(*
SPDX-FileCopyrightText: © 2026 Oleksandr Tiutyk <trofimich@gmail.com>
SPDX-License-Identifier: MIT
License: https://opensource.org/license/mit
*)

(*!
<summary>Executes TryActivity and recovers via an optional CatchActivity when TryActivity raises an exception.</summary>
<description>
When TryActivity throws a non-terminal exception and CatchActivity is configured, synchronous diagnostics are
passed to CatchActivity.CaptureException before starting CatchActivity. Terminal allocation failures and
exceptions when CatchActivity is 0 (or thrown by CatchActivity itself) propagate to the parent. Resetting
resets both TryActivity and CatchActivity back to PASSIVE_READY and clears CurrentActivity. Catch startup
does not wait for asynchronous cleanup in the failed try branch. The recovery implementation must use
independent resources or explicitly coordinate cleanup completion before reusing a shared resource.
A failed try branch is not automatically reset before catch. After the composite finishes, RequestReset
provides the ordinary path for driving pending cancellation/reset work before a fresh run.
</description>
*)

{attribute 'no_explicit_call' := 'do not call this function block directly'}
{attribute 'enable_dynamic_creation'}
FUNCTION_BLOCK TryCatchActivity EXTENDS ExclusiveCompositeActivity
	IMPLEMENTS ITryCatchActivity, TOF_Core.IConfigurationSerializable
VAR_STAT
	{attribute 'hide'}
	_ClassName : STRING := __POUNAME();
END_VAR
VAR
	{attribute 'OPC.UA.DA' := '0'}
	_TryActivity : IActivity;

	{attribute 'OPC.UA.DA' := '0'}
	_CatchActivity : ICatchActivity;

	{attribute 'OPC.UA.DA' := '0'}
	_CurrentActivity : IActivity;
END_VAR

(*!
<summary>Returns the optional recovery activity executed when TryActivity raises an exception.</summary>
*)
{attribute 'monitoring' := 'call'}
PROPERTY FINAL CatchActivity : ICatchActivity
GET
CatchActivity := _CatchActivity;
END_GET
END_PROPERTY

(*!
<summary>Borrows the initialized class name used in diagnostics.</summary>
<description>
Returns initialized metadata storage without allocation. Callers must not modify the returned string.
Derived function blocks must use distinct initialized static storage when overriding this metadata.
</description>
*)
{attribute 'monitoring' := 'call'}
PROPERTY ClassName : REFERENCE TO STRING
GET
ClassName REF= _ClassName;
END_GET
END_PROPERTY

(*!
<summary>Configures the required TryActivity and optional CatchActivity.</summary>
<description>
Permitted only in PASSIVE_READY. Validates all supplied references before mutating state.
</description>
<param name="tryActivity">Required primary activity to execute.</param>
<param name="catchActivity">Optional recovery activity invoked when tryActivity fails, or 0.</param>
*)
METHOD Configure
VAR_INPUT
	tryActivity : IActivity;
	catchActivity : ICatchActivity;
END_VAR
VAR
END_VAR
ValidateChildActivityAttachment(childActivity := tryActivity, argumentName := 'tryActivity');

IF catchActivity <> 0 THEN
	ValidateChildActivityAttachment(childActivity := catchActivity, argumentName := 'catchActivity');

	IF catchActivity.SelfAddress = tryActivity.SelfAddress THEN
		WorkflowExceptions.ThrowWorkflowConfiguration(
			sourceNamespaceName := NamespaceName,
			sourceClassName := ClassName,
			sourcePOUName := __POUNAME(),
			sourcePosition := __POSITION(),
			message := "TryActivity and CatchActivity cannot reference the same activity instance"
		);
	END_IF
END_IF

_TryActivity := tryActivity;
_TryActivity.ParentActivity := THIS^;

_CatchActivity := catchActivity;

IF _CatchActivity <> 0 THEN
	_CatchActivity.ParentActivity := THIS^;
END_IF
END_METHOD

(*!
<summary>Returns the currently active branch (TryActivity or CatchActivity), or 0 when idle.</summary>
*)
{attribute 'monitoring' := 'call'}
PROPERTY FINAL CurrentActivity : IActivity
GET
CurrentActivity := _CurrentActivity;
END_GET
END_PROPERTY

(*!
<summary>Borrows the compiler-initialized library namespace.</summary>
<description>
Borrows storage from the live internal namespace provider. Reacquire references after application
reinitialization or relocation. Treat the reference as read-only; no ownership or synchronization is provided.
</description>
*)
{attribute 'monitoring' := 'call'}
PROPERTY NamespaceName : REFERENCE TO STRING
GET
NamespaceName REF= CurrentNamespace.Name;
END_GET
END_PROPERTY

(*!
<summary>Resets TryActivity and CatchActivity back to PASSIVE_READY and clears CurrentActivity.</summary>
<param name="startResetting">TRUE on the initial call from RequestReset.</param>
*)
METHOD PROTECTED OnResetting : ACTIVITY_RESETTING_STATE
VAR_INPUT
	startResetting : BOOL;
END_VAR
IF _TryActivity <> 0 AND_THEN _TryActivity.State <> WORKFLOW_ELEMENT_STATE.PASSIVE_READY THEN
	IF ResetChildActivity(childActivity := _TryActivity) = ACTIVITY_RESETTING_STATE.WORK_IN_PROGRESS THEN
		OnResetting := ACTIVITY_RESETTING_STATE.WORK_IN_PROGRESS;
		RETURN;
	END_IF
END_IF

IF _CatchActivity <> 0 AND_THEN _CatchActivity.State <> WORKFLOW_ELEMENT_STATE.PASSIVE_READY THEN
	IF ResetChildActivity(childActivity := _CatchActivity) = ACTIVITY_RESETTING_STATE.WORK_IN_PROGRESS THEN
		OnResetting := ACTIVITY_RESETTING_STATE.WORK_IN_PROGRESS;
		RETURN;
	END_IF
END_IF

_CurrentActivity := 0;
OnResetting := ACTIVITY_RESETTING_STATE.WORK_RESET;
END_METHOD

(*!
<summary>Runs TryActivity and transitions to CatchActivity if TryActivity raises a non-terminal exception.</summary>
<param name="startRunning">TRUE on the initial call of a fresh start.</param>
<param name="startResuming">TRUE on the initial call when resuming from suspension.</param>
<param name="haltReason">Receives the active child's HaltReason when halted.</param>
*)
METHOD PROTECTED OnRunning : ACTIVITY_RUNNING_STATE
VAR_INPUT
	startRunning : BOOL;
	startResuming : BOOL;
END_VAR
VAR_OUTPUT
	haltReason : WSTRING(255);
END_VAR
VAR

	exceptionCode : __SYSTEM.ExceptionCode;
	exception : TOF_Core.IException;
END_VAR
IF _TryActivity = 0 THEN
	TOF_Core.Exceptions.ThrowNullReference(
		sourceNamespaceName := NamespaceName,
		sourceClassName := ClassName,
		sourcePOUName := __POUNAME(),
		sourcePosition := __POSITION(),
		variableOrPropertyName := 'TryActivity'
	);
END_IF

IF startRunning OR_ELSE (startResuming AND_THEN _CurrentActivity = 0) THEN
	_CurrentActivity := _TryActivity;
END_IF

IF _CurrentActivity = _TryActivity THEN
	__TRY
		IF startRunning OR_ELSE startResuming THEN
			_CurrentActivity.RequestStart();
		ELSE
			_CurrentActivity.Execute();
		END_IF

		OnRunning := MapChildRunningState(childState := _CurrentActivity.State);

		IF OnRunning = ACTIVITY_RUNNING_STATE.WORK_HALTED THEN
			haltReason := _CurrentActivity.HaltReason;
		END_IF
	__CATCH(exceptionCode)
		TOF_Core.DynamicMemoryManager.RaiseIfAllocationFailed();

		IF _CatchActivity = 0 THEN
			TOF_Core.ExceptionManager.ReThrowLastException(
				exceptionCode := exceptionCode,
				catchPointNamespaceName := NamespaceName,
				catchPointPOUName := __POUNAME(),
				catchPointPosition := __POSITION()
			);
		END_IF

		exception := TOF_Core.ExceptionManager.GetLastException(
			exceptionCode := exceptionCode,
			catchPointNamespaceName := NamespaceName,
			catchPointPOUName := __POUNAME(),
			catchPointPosition := __POSITION()
		);

		// Keep the native wrapper stable while CaptureException may handle another exception.

		IF NOT exception.IsDynamicInstance THEN
			__QUERYINTERFACE(exception.Clone(), exception);
		END_IF

		__TRY
			_CatchActivity.CaptureException(exception := exception);
		__CATCH
			TOF_Core.DynamicMemoryManager.RaiseIfAllocationFailed();
			TOF_Core.ExceptionManager.Throw(exception := exception);
		__ENDTRY

		TOF_Core.DynamicMemoryManager.RaiseIfAllocationFailed();

		_CurrentActivity := _CatchActivity;
		_CurrentActivity.RequestStart();

		OnRunning := MapChildRunningState(childState := _CurrentActivity.State);

		IF OnRunning = ACTIVITY_RUNNING_STATE.WORK_HALTED THEN
			haltReason := _CurrentActivity.HaltReason;
		END_IF
	__ENDTRY
ELSIF _CurrentActivity <> 0 AND_THEN _CatchActivity <> 0 AND_THEN _CurrentActivity.SelfAddress = _CatchActivity.SelfAddress THEN
	IF startResuming THEN
		_CurrentActivity.RequestStart();
	ELSE
		_CurrentActivity.Execute();
	END_IF

	OnRunning := MapChildRunningState(childState := _CurrentActivity.State);

	IF OnRunning = ACTIVITY_RUNNING_STATE.WORK_HALTED THEN
		haltReason := _CurrentActivity.HaltReason;
	END_IF
END_IF
END_METHOD

(*!
<summary>Stops the currently active try or catch branch on cancel or suspend.</summary>
<param name="startCancelling">TRUE on the initial call from RequestCancel.</param>
<param name="startSuspending">TRUE on the initial call from RequestSuspend.</param>
<param name="haltReason">Receives the active branch's HaltReason if it halts while stopping.</param>
*)
METHOD PROTECTED OnStopping : ACTIVITY_STOPPING_STATE
VAR_INPUT
	startCancelling : BOOL;
	startSuspending : BOOL;
END_VAR
VAR_OUTPUT
	haltReason : WSTRING(255);
END_VAR
IF _CurrentActivity = 0 THEN
	OnStopping := ACTIVITY_STOPPING_STATE.WORK_STOPPED;
	RETURN;
END_IF

IF NOT _CurrentActivity.Busy THEN
	IF startCancelling AND_THEN _CurrentActivity.State = WORKFLOW_ELEMENT_STATE.PASSIVE_SUSPENDED THEN
		_CurrentActivity.RequestCancel(reason := _CancelReason);
	END_IF

	OnStopping := MapChildStoppingState(childState := _CurrentActivity.State);

	IF OnStopping = ACTIVITY_STOPPING_STATE.WORK_HALTED THEN
		haltReason := _CurrentActivity.HaltReason;
	END_IF

	RETURN;
END_IF

IF startCancelling THEN
	_CurrentActivity.RequestCancel(reason := _CancelReason);
ELSIF startSuspending THEN
	_CurrentActivity.RequestSuspend();
ELSE
	_CurrentActivity.Execute();
END_IF

OnStopping := MapChildStoppingState(childState := _CurrentActivity.State);

IF OnStopping = ACTIVITY_STOPPING_STATE.WORK_HALTED THEN
	haltReason := _CurrentActivity.HaltReason;
END_IF
END_METHOD

(*!
<summary>Reports the size of this concrete function block instance in bytes.</summary>
<description>
Reports the instance layout rather than dynamic allocations owned by its fields. A derived function block
with a different layout must override this property; the value does not grant disposal rights.
</description>
*)
{attribute 'monitoring' := 'call'}
PROPERTY SelfSize : ULINT
GET
SelfSize := XSIZEOF(THIS^);
END_GET
END_PROPERTY

(*!
<summary>Returns the primary activity executed by this composite.</summary>
*)
{attribute 'monitoring' := 'call'}
PROPERTY FINAL TryActivity : IActivity
GET
TryActivity := _TryActivity;
END_GET
END_PROPERTY

(*!
<summary>Writes the configuration fields for this object.</summary>
<description>Borrows the writer for this call. A failure invalidates the current output document.</description>
*)
METHOD Serialize
VAR_INPUT
	writer : TOF_Core.IConfigurationWriter;
END_VAR
Workflows.WriteConfigurationHeader(writer := writer, source := THIS^, displayName := Name, scope := THIS^);
Workflows.WriteConfigurationObject(writer := writer, name := 'tryActivity', source := _TryActivity);

IF _CatchActivity <> 0 THEN
	Workflows.WriteConfigurationObject(writer := writer, name := 'catchActivity', source := _CatchActivity);
END_IF
END_METHOD

(*!
<summary>Restores this fresh instance from its configuration object.</summary>
<description>
The reader, document node and deserialization context are borrowed for this call.
On failure discard the partial instance.
</description>
<param name="reader">Active configuration reader.</param>
<param name="node">Configuration node for this activity.</param>
<param name="context">Active configuration deserialization context providing workflow reconstruction services.</param>
*)
METHOD Deserialize
VAR_INPUT
	reader : TOF_Core.IConfigurationReader;
	node : TOF_Core.CONFIGURATION_NODE;
	context : TOF_Core.IConfigurationDeserializationContext;
END_VAR
VAR
	loader : IWorkflowLoader;
END_VAR
loader := WorkflowConfigurationSerializer.ResolveWorkflowLoader(context := context);
Workflows.ReadConfigurationHeader(reader := reader, node := node, target := THIS^, scope := THIS^);

Configure(
	tryActivity := Workflows.ReadActivity(loader := loader, node := reader.GetField(node := node, name := 'tryActivity')),
	catchActivity := Workflows.ReadCatchActivity(loader := loader, node := reader.FindField(node := node, name := 'catchActivity'))
);
END_METHOD

END_FUNCTION_BLOCK

(* stored: Version 1.1.0.1
   POU TryCatchActivity: Id {a1c6778a-1c1f-42dd-a420-c513f7979378}, SpecialFunc None
   Folder Overriden methods: Id {5198ec74-8b1a-4d40-bf51-2490efda6192}
   Property CatchActivity: Id {d45db91b-6e3c-4d25-88ad-eccd861a1235}
   Get Get: Id {d47a176f-7515-4853-bd3a-48f4103cee47}
   Property ClassName: Id {fdfdec0c-6bcb-49f1-bea5-0a524cb226e3}
   Get Get: Id {0d4ca4db-bcfb-4d1e-bfc1-64b96a5d7f54}
   Method Configure: Id {1ad8b2fa-0f3e-40cb-907d-1c905fa035da}
   Property CurrentActivity: Id {882195bd-d9d1-4458-ab34-d7d9d29e51f1}
   Get Get: Id {2f22007f-b61b-46eb-b0f7-86bd74729b31}
   Property NamespaceName: Id {e11525f6-0bdd-472c-8148-75ceee244093}
   Get Get: Id {efaef8de-4de6-4c21-a478-c15946922349}
   Method OnResetting: Id {5b92043f-7a56-4812-8b93-2f93c74a1504}
   Method OnRunning: Id {ca2f10c4-f86d-4e87-bfe8-d64bbb3b6bc6}
   Method OnStopping: Id {3ff4c539-5cf6-4ae8-9712-0a7f4b6fdb99}
   Property SelfSize: Id {e3dcfcd8-e5b6-434c-b73b-40d8ae840636}
   Get Get: Id {7018bfdf-c2ce-492d-a525-6244d2e5d50f}
   Property TryActivity: Id {a258f937-76f3-47db-be03-89bec51ed17e}
   Get Get: Id {c24798e4-9b45-4cdf-b41a-9fccd6b4f85b}
   Method Serialize: Id {9c60f75b-d656-44ab-a4a1-542acc44035f}
   Method Deserialize: Id {804f42e5-7bca-4936-a972-344bb4532c66} *)
